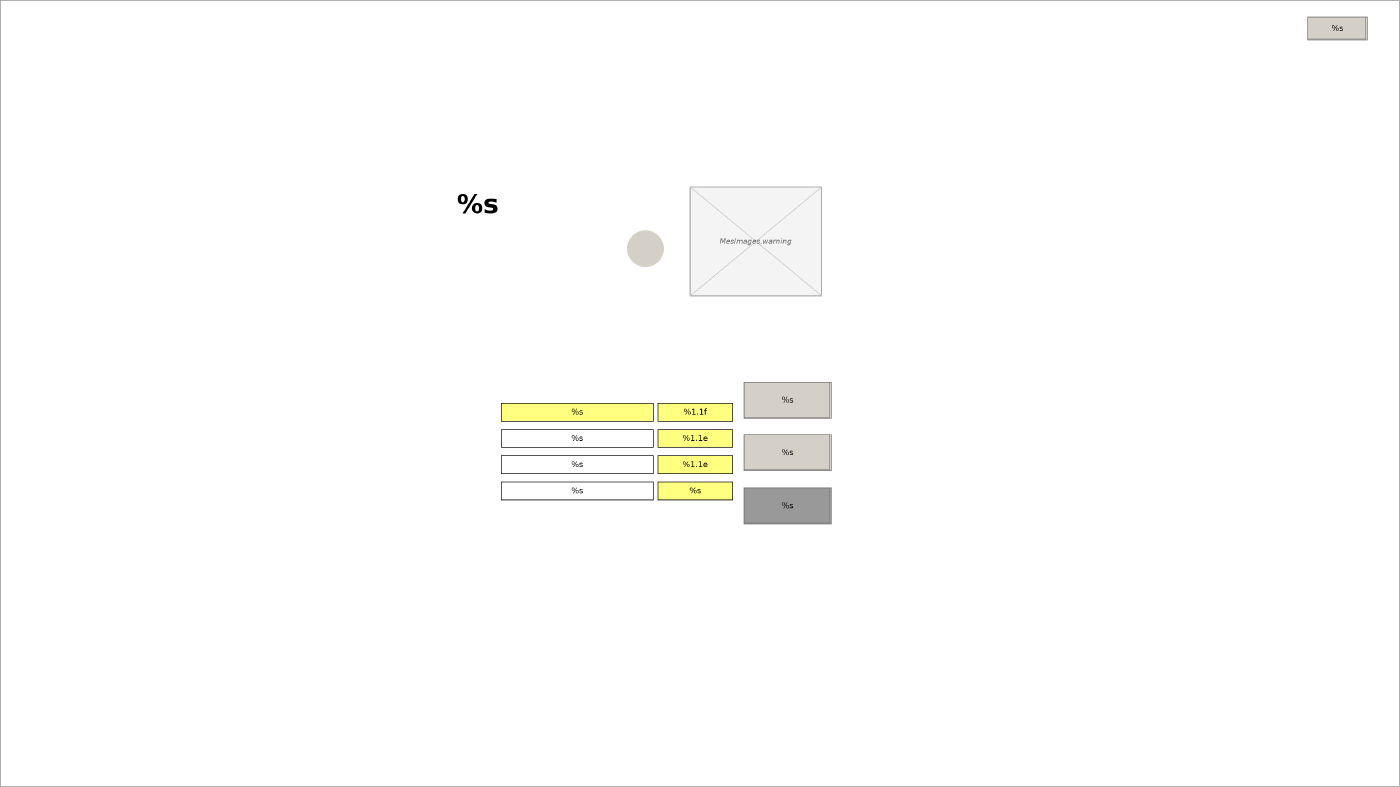
VISUALIZATION VISU_VANNE_ASS_H_MANU  // 1920x1080
VAR_IN_OUT
	m_Input_Vanne:		BLOCK_VVAT_650_NO;
	m_Input_State_Manu:	BOOL;
END_VAR
    Button (1793,23 82x32), "%s", text list: 'TextList_Basiques', text index: 8
        OnMouseClick: change screen: Previous 
        OnMouseClick: execute { .VISU_INDEX_MANU := 0; }
    Polygon (0,0), colour toggle: m_Input_VANNE.STATE_Lam
    Rectangle (573,246 165x68), "%s", text variable: m_Input_VANNE.MNEMO
    Polygon (0,0), colour toggle: m_Input_VANNE.STATE_On, invisible if: NOT (m_Input_VANNE.STATE_Off OR m_Input_VANNE.STATE_On)
    Ellipse (860,316 50x50), colour toggle: m_Input_VANNE.STATE_Ok
    Image (946,256 181x150), invisible if: NOT m_Input_VANNE.STATE_Nok, image: MesImages.warning
    Button (1020,524 120x50), "%s", input disabled if: NOT m_Input_Vanne.AUTOR_On_IHM OR NOT .PRG_USER.ACTU_USER.MAINTENANCE, text list: 'TextList_VVAT_3P', text index: 0
        toggle m_Input_Vanne.M_On
    Button (1020,596 120x50), "%s", input disabled if: NOT m_Input_Vanne.AUTOR_Off_IHM OR NOT .PRG_USER.ACTU_USER.MAINTENANCE, text list: 'TextList_VVAT_3P', text index: 1
        toggle m_Input_Vanne.M_Off
    Button (1020,669 120x50), "%s", input disabled if: NOT m_Input_Vanne.AUTOR_Lam_IHM OR NOT .PRG_USER.ACTU_USER.MAINTENANCE, text list: 'TextList_VVAT_3P', text index: 2
        toggle m_Input_Vanne.M_Lam
    RoundedRectangle (687,553 209x25), "%s", invisible if: NOT m_Input_Vanne.PRM_Mode, input disabled if: NOT .PRG_USER.ACTU_USER.MAINTENANCE OR NOT m_Input_State_Manu OR NOT m_Input_Vanne.PRM_Mode, text list: 'TextList_VVAT_650_ETHERCAT', text index: 8
        OnMouseClick: toggle m_Input_Vanne.PRM_Mode
    RoundedRectangle (687,553 209x25), "%s", invisible if: m_Input_Vanne.PRM_Mode, input disabled if: NOT .PRG_USER.ACTU_USER.MAINTENANCE OR NOT m_Input_State_Manu OR m_Input_Vanne.PRM_Mode, text list: 'TextList_VVAT_650_ETHERCAT', text index: 7
        OnMouseClick: toggle m_Input_Vanne.PRM_Mode
    RoundedRectangle (687,589 209x25), "%s", invisible if: NOT m_Input_Vanne.PRM_Mode, text list: 'TextList_VVAT_650_ETHERCAT', text index: 4
    RoundedRectangle (687,625 209x25), "%s", invisible if: NOT m_Input_Vanne.PRM_Mode, text list: 'TextList_VVAT_650_ETHERCAT', text index: 5
    RoundedRectangle (687,661 209x25), "%s", invisible if: NOT m_Input_Vanne.PRM_Mode, text list: 'TextList_VVAT_650_ETHERCAT', text index: 6
    RoundedRectangle (902,661 103x25), "%s", text variable: m_Input_Vanne.PRM_Tim_W_Pr, invisible if: NOT m_Input_Vanne.PRM_Mode, input disabled if: NOT m_Input_Vanne.PRM_Mode
        OnMouseClick: write the text variable via Edit
    RoundedRectangle (902,625 103x25), "%1.1e", text variable: m_Input_Vanne.PRM_W_Pr_HI, invisible if: NOT m_Input_Vanne.PRM_Mode, input disabled if: NOT m_Input_Vanne.PRM_Mode
        OnMouseClick: write the text variable via InputWithLimits, min 0, max 1000
    RoundedRectangle (902,589 103x25), "%1.1e", text variable: m_Input_Vanne.PRM_W_Pr_LO, invisible if: NOT m_Input_Vanne.PRM_Mode, input disabled if: NOT m_Input_Vanne.PRM_Mode
        OnMouseClick: write the text variable via InputWithLimits, min 0, max 1000
    RoundedRectangle (902,553 103x25), "%1.1e", text variable: m_Input_Vanne.PRM_Pression, invisible if: NOT m_Input_Vanne.PRM_Mode, input disabled if: NOT m_Input_Vanne.PRM_Mode
        OnMouseClick: write the text variable via InputWithLimits, min 0, max 1000
    RoundedRectangle (902,553 103x25), "%1.1f", text variable: m_Input_Vanne.PRM_Position, invisible if: m_Input_Vanne.PRM_Mode, input disabled if: m_Input_Vanne.PRM_Mode
        OnMouseClick: write the text variable via InputWithLimits, min 0, max 100
END_VISUALIZATION

(* stored: Version 1.1.0.1, ProductVersion 3.1.4026.18
   Visu VISU_VANNE_ASS_H_MANU: Id {3ada4f15-3bdd-430e-bf2d-f0a05526c74c} *)
